// SIMATIC S7-200 SMART project (STEP 7-Micro/WIN SMART), CPU SR30

SYMBOL_TABLE System Symbols
Clock_1s         SM0.5    // Clock pulse that is ON for 0.5 s, OFF for 0.5 s, for a duty cycle time of 1 s.
END_SYMBOL_TABLE

ORGANIZATION_BLOCK MAIN:OB1
TITLE=Program Comments
BEGIN
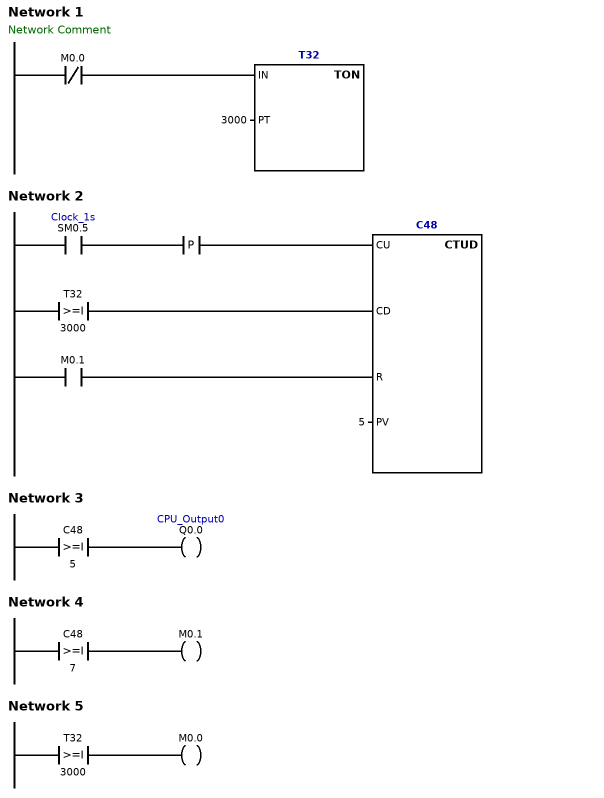
Network 1
// Network Comment
LDN    M0.0
TON    T32, 3000
Network 2
LD     Clock_1s:SM0.5
EU
LDW>=  T32, 3000
LD     M0.1
CTUD   C48, 5
Network 3
LDW>=  C48, 5
=      CPU_Output0:Q0.0
Network 4
LDW>=  C48, 7
=      M0.1
Network 5
LDW>=  T32, 3000
=      M0.0
END_ORGANIZATION_BLOCK
